ABB RAPID module: Module_no_1.mod

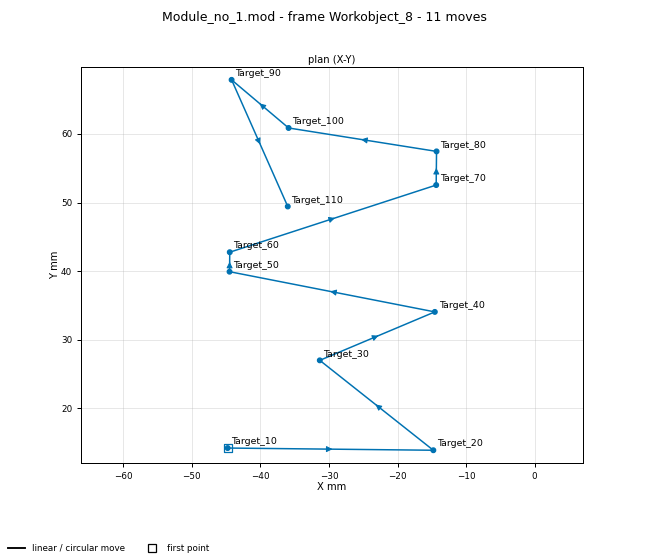
[picture p0: tool path of Module_no_1.mod in frame Workobject_8, 11 of 11 moves have a stored position in this frame; points joined in program order, loops and branches not executed]
MODULE Module1
        CONST robtarget Target_10:=[[-44.771402545,14.191657604,-20],[0,0.710877818,0.703315525,0],[0,0,0,0],[9E+09,9E+09,9E+09,9E+09,9E+09,9E+09]];
    CONST robtarget Target_20:=[[-14.773118193,13.870821271,-20],[0,0.710877818,0.703315525,0],[0,0,0,0],[9E+09,9E+09,9E+09,9E+09,9E+09,9E+09]];
    CONST robtarget Target_30:=[[-31.335839797,26.982701879,-20],[0,0.710877818,0.703315525,0],[0,0,0,0],[9E+09,9E+09,9E+09,9E+09,9E+09,9E+09]];
    CONST robtarget Target_40:=[[-14.557312981,34.048667269,-20],[0,0.710877818,0.703315525,0],[0,0,0,0],[9E+09,9E+09,9E+09,9E+09,9E+09,9E+09]];
    CONST robtarget Target_50:=[[-44.496317473,39.912186607,-20],[0,0.710877818,0.703315525,0],[0,0,0,0],[9E+09,9E+09,9E+09,9E+09,9E+09,9E+09]];
    CONST robtarget Target_60:=[[-44.465902189,42.756023963,-20],[0,0.710877818,0.703315525,0],[0,0,0,0],[9E+09,9E+09,9E+09,9E+09,9E+09,9E+09]];
    CONST robtarget Target_70:=[[-14.359463909,52.547609286,-20],[0,0.710877818,0.703315525,0],[0,0,0,0],[9E+09,9E+09,9E+09,9E+09,9E+09,9E+09]];
    CONST robtarget Target_80:=[[-14.306943002,57.458328434,-20],[0,0.710877818,0.703315525,0],[0,0,0,0],[9E+09,9E+09,9E+09,9E+09,9E+09,9E+09]];
    CONST robtarget Target_100:=[[-35.884644867,60.874287478,-20],[0,0.710877818,0.703315525,0],[0,0,0,0],[9E+09,9E+09,9E+09,9E+09,9E+09,9E+09]];
    CONST robtarget Target_90:=[[-44.197062731,67.892586365,-20],[0,0.710877818,0.703315525,0],[0,0,0,0],[9E+09,9E+09,9E+09,9E+09,9E+09,9E+09]];
    CONST robtarget Target_110:=[[-36.007108096,49.423942341,-20],[0,0.710877818,0.703315525,0],[0,0,0,0],[9E+09,9E+09,9E+09,9E+09,9E+09,9E+09]];
!***********************************************************
    !
    ! M?dulo:  Module1
    !
    ! Descripción:
    !   <Introduzca la descripción aquí>
    !
    ! Autor: Andres
    !
    ! Versión: 1.0
    !
    !***********************************************************


    !***********************************************************
    !
    ! Procedimiento Main
    !
    !   Este es el punto de entrada de su programa
    !
    !***********************************************************
    PROC main()
        !Add your code here
    ENDPROC
    PROC Path_10()
        MoveL Target_10,v1000,z100,CualquierCosa\WObj:=Workobject_8;
        MoveL Target_20,v1000,z100,CualquierCosa\WObj:=Workobject_8;
        MoveL Target_30,v1000,z100,CualquierCosa\WObj:=Workobject_8;
        MoveL Target_40,v1000,z100,CualquierCosa\WObj:=Workobject_8;
        MoveL Target_50,v1000,z100,CualquierCosa\WObj:=Workobject_8;
        MoveL Target_60,v1000,z100,CualquierCosa\WObj:=Workobject_8;
        MoveL Target_70,v1000,z100,CualquierCosa\WObj:=Workobject_8;
        MoveL Target_80,v1000,z100,CualquierCosa\WObj:=Workobject_8;
        MoveL Target_100,v1000,z100,CualquierCosa\WObj:=Workobject_8;
        MoveL Target_90,v1000,z100,CualquierCosa\WObj:=Workobject_8;
        MoveL Target_110,v1000,z100,CualquierCosa\WObj:=Workobject_8;
    ENDPROC
ENDMODULE
